(* CODESYS project PresentazioneGIT
   Author: Francesco
   Title: M262 Slave Modbus e ServerOPC_UA
   Version: 0.0.0.0

Project tree, tasks and I/O mapping:
  MyController : TM262L10MESE8T, Schneider Electric, order no. TM262L10MESE8T, version 5.2.8.12
      settings: Enable OPC-UA Server = True; NTP_SERVERENA = False; InterfaceUsedByDhcpSize = 0
    application Application
      libraries: HttpHandling, 1.3.6.0 (Schneider Electric); SysTimeRtc, * (System); TcpUdpCommunication, 2.3.0.0 (Schneider Electric); SysMem, * (System); VisuDialogs, * (System); IecRtsServices, 1.0.5.0 (Schneider Electric); TimeSync, 1.1.7.0 (Schneider Electric); CertificateHandling, 1.2.1.0 (Schneider Electric); CAA File, * (CAA Technical Workgroup)
      task MAST (cyclic, interval 20 ms, priority 15, watchdog 60 ms x 2) calls POU_API_Manuale
      program Certificate_Handling [ST]
      Prog_MatteoLoda/
        data type DUT_result_GET
        global variables GVL_opcua
        global variables PersistentVars
        program POU_API_Manuale [ST]: ACT_Gestione_String_Lettura, New_action
        Symbols
    Diagnostic
    Machine Assistant
    Message Logger
    COM_Bus : COM Bus - TMS, Schneider Electric, version 5.2.8.12
        settings: Network Address = [199, 169, 2, 0]
    DI : Digital Inputs, Schneider Electric, version 5.2.8.12
        input  ibDI_IB0 : BYTE  // IB0
        input  ibDI_IB1 : BYTE  // IB1
    DQ : Digital Outputs, Schneider Electric, version 5.2.8.12
        output q0 : BOOL  // QB0.Q0
        output q1 : BOOL  // QB0.Q1
        output q2 : BOOL  // QB0.Q2
        output q3 : BOOL  // QB0.Q3
        unmapped channels: QB0, QB1
    Ethernet_2 : ETH2, Schneider Electric, version 5.2.8.12
        settings: IPAddress = [192, 168, 8, 19]; SubnetMask = [255, 255, 255, 0]; WebServer = TRUE; FTP Server = TRUE; SoMachine Protocol = TRUE; Modbus Server = TRUE; NetManage Protocol = TRUE; SNMP protocol = TRUE; WebVisu protocol = TRUE; Secured Web Server = TRUE; Remote Connection = TRUE
    Ethernet_Sercos : ETH1, Schneider Electric, version 5.2.8.12
        settings: IPAddress = [192, 168, 1, 91]; SubnetMask = [255, 255, 255, 0]; GatewayAddress = [192, 168, 1, 1]; WebServer = TRUE; FTP Server = TRUE; SoMachine Protocol = TRUE; Modbus Server = TRUE; NetManage Protocol = TRUE; SNMP protocol = TRUE; WebVisu protocol = TRUE; Secured Web Server = TRUE; Remote Connection = TRUE
    IO_Bus : IO bus - TM3, Schneider Electric, version 5.2.8.12
    Serial_Line : Serial line, Schneider Electric, version 5.2.8.12
  5ce3da45-db07-42e7-a21c-a00fff4ed8f6|C:\Users\sesa18348\Downloads\connectivity_1024_768.jpg
  text list GlobalTextList
  function GetCompany [ST]
  function GetTextProperty2 [ST]
  function GetTextProperty [ST]
  function GetTitle [ST]
  function GetVersion [ST]
  function GetVersionProperty [ST]
*)

// MyController/Application/Prog_MatteoLoda/DUT_result_GET
TYPE DUT_result_GET :
STRUCT
	valore:  STRING;
	timestamp:  STRING;
END_STRUCT
END_TYPE

// MyController/Application/Prog_MatteoLoda/GVL_opcua
VAR_GLOBAL
	

scada_data_ora_start : STRING  ;  // data ora start , arriva da scada expert con questo formato : '2023-06-20T04:44:30Z'
scada_data_ora_end : STRING  ; // data ora start , arriva da scada expert con questo formato : '2023-06-20T04:45:00Z' 

Result_Get_value: ARRAY[0..19] OF STRING;
Result_Get_timestamp: ARRAY[0..19] OF STRING;
puntatore_GET: INT;


reset_n_richieste : BOOL ;


ind_IP_Dominio : STRING ; // ip ricevuto da funzione dns
x_dns_OK: BOOL; // dns ok significa anche internet ok
x_dns_ERR: BOOL; // dns err significa anche errore internet
//x_Ping_OK: BOOL;
//x_Ping_ERR: BOOL;
result_HTTP: STRING(INT#15); 
http_client_state			: SE_HTTP.ET_State; // Idle=0, Connecting=10, Connected=20, SendingRequest=30 , Disconnecting=40 ,ResponseAvailable=50 ,Error=-10	
n_dns_ERR: UDINT;

gx_StartCertHandling : bool;


END_VAR

// MyController/Application/Prog_MatteoLoda/PersistentVars

VAR_GLOBAL PERSISTENT RETAIN
	






diag_n_richieste_OK : UDINT ;
diag_n_richieste_ERR : UDINT ;

time_polling : INT ; // tempo base ms












END_VAR

// MyController/Application/Prog_MatteoLoda/POU_API_Manuale
PROGRAM POU_API_Manuale
VAR CONSTANT
String_Unit_ID : ARRAY[0..19] OF STRING := ['formula_ids=2925', 'unit_ids=36389', 'unit_ids=36384', 'unit_ids=36387', 'formula_ids=2931', 'unit_ids=36342', 'unit_ids=36337', 'unit_ids=36340', 'formula_ids=2929', 'unit_ids=36351', 'unit_ids=36346', 'unit_ids=36349', 'formula_ids=2930', 'unit_ids=36371', 'unit_ids=36366', 'unit_ids=36369', 'formula_ids=2928', 'unit_ids=36380', 'unit_ids=36375', 'unit_ids=36378'] ;
END_VAR

VAR
String_Resource: STRING(200);

// Lib usate in questa Demo : SE_HTTP ( x funzioni di connessione e scritture https )
// Lib usate in questa Demo : TCPUDP ( x funzione dns )
// Lib usate in questa Demo : SysTimeRtc ( x funzione timestamp )		
FB_DNSCLIENT				: TCPUDP.FB_DnsClient;			// dichiarazione dell'FB DNS per recupero indirizzo ip del server
FB_HTTP_CLIENT				: SE_HTTP.FB_HttpClient;		// dichiarazione dell'FB CLIENT per connessione , scrittura dati e disconnessione
PARAM_ConnectToServer		: SE_HTTP.TlsSettings;			// ingresso dell'FB : FB_HTTP_CLIENT.ConnectToServer	

Get_Result: SE_HTTP.ET_Result;

Get_result_Msg : STRING ;
Get_Additional_Header: STRING;
Get_Response_Buffer : STRING(5000); // ricezione dati  , per export opcua max(254)
get_error: BOOL;
Get_Strart_request: BOOL;
Get_String_Resource: STRING(SE_HTTP.GPL.Gc_uiMaxLengthOfResource);
FB_PING: TCPUDP.FB_Ping;
ResultPing: STRING(80);
xResultPing: BOOL;
xExecPing : BOOL ;
xResultConnect: SE_HTTP.ET_Result;
temp_string: STRING(1000);
key: STRING(INT#5);
key_stamp: STRING(INT#9);
i: INT;
b: INT;
c: INT;
key2: STRING(INT#1);
a: INT;

x: INT;

	sts: INT;
	sts_prec: INT;
	
	FB_Rit_Start_Polling: TON;
	Dns_leggi_ip: BOOL;
cmd_Reset_Disconnect: BOOL;
cmd_CONNESSIONE: BOOL;
	n_bcd: BYTE;
	FB_NTP: TIMS.FB_SntpClient;
	F_Blink_01: BLINK;
	ntp_manual: BOOL;
	


x_Ping_OK  : BOOL;
x_Ping_ERR : BOOL;

	xNtp_first_time: BOOL;
	xNtp_first_time_done: BOOL;

ritardo_primo_ntp : TON;
impulso_primo_ntp : TP;

ritarda_CertHandling : TON;
END_VAR


// esempio string richiesta GET
// '/api/v2/export/?start=2023-06-20T04:44:30Z&end=2023-06-20T04:45:00Z&unit_ids=36389'
String_Resource := CONCAT('/api/v2/export/?start=',scada_data_ora_start) ; // prepara string get
String_Resource := CONCAT(String_Resource,'&end=') ;// prepara string get
String_Resource := CONCAT(String_Resource,scada_data_ora_end) ;// prepara string get
String_Resource := CONCAT(String_Resource,'&') ;// prepara string get
String_Resource := CONCAT(String_Resource,String_Unit_ID[puntatore_GET]) ;// prepara string get


// parametri per FB connessione
PARAM_ConnectToServer.etProtocol 		:= TCPUDP.ET_TlsProtocol.TLSv13 ;  				// impostazione Parametri per FB seguente 
PARAM_ConnectToServer.etCertVerifyMode 	:= TCPUDP.ET_CertVerifyMode.TrustedOnly  ;	 	// impostazione Parametri per FB seguente

// parametri per FB GET
//Get_String_Resource := '/api/v2/export/?start=2023-06-20T04:44:30Z&end=2023-06-20T04:45:00Z&unit_ids=36389'   ; // 
Get_String_Resource := String_Resource  ; // 
Get_Additional_Header :=  'Authorization: Basic emVudHJpeDpyaXZlcmxha2U='   ; // 'Authorization: Basic b3BlcmF0b3I6ZGU0NzU5MzE='  codificato in base64
	



//---------------------------------------------------------------------------------------------------------------------

// time_polling
IF time_polling<5 THEN // timepolling è usato come ritardo tra richieste , tempo min 5 ms
	time_polling := 5 ; // tempo min 5 ms
END_IF
FB_Rit_Start_Polling(
	IN:=NOT Dns_leggi_ip , 
	PT:= INT_TO_TIME(time_polling), 
	Q=> , 
	ET=> );
IF 	FB_Rit_Start_Polling.Q THEN
	Dns_leggi_ip:=TRUE;
END_IF

//---------------------------------------------------------------------------------------------------------------------

FB_DNSCLIENT(
	i_xEnable			:=  Dns_leggi_ip, 
	i_xExecute			:=  FB_DNSCLIENT.q_xActive AND FB_DNSCLIENT.q_xReady, 
	i_sDnsServerIP		:= '8.8.8.8', // dns di google
	i_uiDnsServerPort	:= , 
	i_sDomainName		:=  'ehp-data.com',  // dominio
	q_xActive			=> , 
	q_xReady			=> , 
	q_xBusy				=> , 
	q_xDone				=> x_dns_OK, 
	q_xError			=> x_dns_ERR, 
	q_etResult			=> , 
	q_sResultMsg		=> , 
	q_uiNumberOfIpAddresses	=> , 
	q_astDnsAddressInfo		=> ); // in questo (.q_astDnsAddressInfo[0].sIpAddress) l'indirizzo IP del server
		

IF FB_DNSCLIENT.q_xDone THEN
	ind_IP_Dominio := FB_DNSCLIENT.q_astDnsAddressInfo[0].sIpAddress	;
	xExecPing := TRUE ;

END_IF
IF FB_DNSCLIENT.q_xError THEN
	Dns_leggi_ip := FALSE ;
	n_dns_ERR := n_dns_ERR +1 ;
END_IF


	
// se abilito il ping il polling ritarda causa esecuzione del ping
FB_PING(
	i_xExecute:= xExecPing, 
	i_sDeviceIP:= ind_IP_Dominio , // '135.181.0.23'
	i_timTimeout:= T#5S, 
	q_xBusy=> , 
	q_xDone=> x_Ping_OK, 
	q_xError=> x_Ping_ERR, 
	q_etResult=> , 
	q_sResultMsg=> ResultPing);

IF x_Ping_OK THEN
	gx_StartCertHandling:=TRUE;
END_IF
ritarda_CertHandling(in:=gx_StartCertHandling, pt:=T#500MS);
IF ritarda_CertHandling.Q THEN
	Certificate_Handling();
END_IF


//---------------------------------------------------------------------------------------------------------------------
IF FB_DNSCLIENT.q_xDone THEN // x_Ping_OK
	cmd_CONNESSIONE := TRUE ;
END_IF
http_client_state :=  FB_HTTP_CLIENT.State ;

IF cmd_CONNESSIONE AND FB_HTTP_CLIENT.State = SE_HTTP.ET_State.Idle THEN 			
	FB_HTTP_CLIENT.ConnectToServer(
		i_sServerIP			:= ind_IP_Dominio , // Indirizzo_IP_server   '135.181.0.23' 
		i_uiServerPort		:= 443 , //443
		i_xUseTls			:= TRUE , // true con port 443 , false per port 80
		i_stTlsSettings		:= PARAM_ConnectToServer, 
		q_xError	=> , 
		q_etResult	=>  xResultConnect, 
		q_sResultMsg=> );
END_IF

IF FB_HTTP_CLIENT.State=SE_HTTP.ET_State.Connected THEN
	FB_HTTP_CLIENT.Get( 
		i_sResource := Get_String_Resource ,
		i_sHost:= 'ehp-data.com' ,// ehp-data.com
		i_anyAdditionalHeader:= Get_Additional_Header, // string Header    'Authorization: Basic b3BlcmF0b3I6ZGU0NzU5MzE='
		i_anyResponseBuffer:= Get_Response_Buffer, // string_xy.000 // ricezione dati
		q_xError=> get_error, 
		q_etResult=> Get_Result , 
		q_sResultMsg=> Get_result_Msg );	
END_IF


ACT_Gestione_String_Lettura();




//---------------------------------------------------------------------------------------------------------------------
IF cmd_Reset_Disconnect OR FB_HTTP_CLIENT.State = SE_HTTP.ET_State.Error THEN
	FB_HTTP_CLIENT.DisconnectFromServer(
		q_xError=> , 
		q_etResult=> , 
		q_sResultMsg=> );
	FB_HTTP_CLIENT.Reset();
	cmd_Reset_Disconnect := FALSE ;
	get_error := FALSE ;
	Dns_leggi_ip := FALSE ;
	xExecPing := FALSE ;
	cmd_CONNESSIONE := FALSE ;
	Get_Strart_request := FALSE ;
	Get_Response_Buffer:='';
	Get_Additional_Header:='';
	Get_result_Msg:='';
	puntatore_GET := puntatore_GET +1 ;
	IF puntatore_GET>19 THEN
		puntatore_GET:=0;
	END_IF
END_IF



n_bcd := int_to_bcd(puntatore_GET); // sposto valore puntatore in uscite plc formato bcd
q0:= n_bcd.0 ; // uscita plc
q1:= n_bcd.1 ;// uscita plc
q2:= n_bcd.2 ;// uscita plc
q3:= n_bcd.3 ;// uscita plc



IF reset_n_richieste THEN
	diag_n_richieste_OK := 0 ;
	diag_n_richieste_ERR := 0;
	n_dns_ERR:=0;
	reset_n_richieste := FALSE ;
END_IF

F_Blink_01(ENABLE:=TRUE , TIMELOW:=T#10M , TIMEHIGH:=T#5S , OUT=> );

ritardo_primo_ntp(IN:= NOT xNtp_first_time_done, PT:= T#30S, Q=> , ET=> );
impulso_primo_ntp(IN:= ritardo_primo_ntp.Q, PT:= T#1S, Q=> xNtp_first_time, ET=> );
IF xNtp_first_time THEN
	xNtp_first_time_done:=TRUE;
END_IF

FB_NTP.i_stTimeRequest.i_sServerIp := '95.217.220.251' ;
FB_NTP.i_stTimeRequest.i_timServerTimeOut := T#3000MS;
FB_NTP(
	i_xEnable:= F_Blink_01.OUT OR ntp_manual OR xNtp_first_time, //
	i_xExecute:= FB_NTP.q_xActive AND FB_NTP.q_xReady, 
	i_xSyncRtc:= TRUE, 
	i_diTimeZone:= , 
	i_uiMaxRtcOffset:= , 
	i_stTimeRequest:= , 
	q_xActive=> , 
	q_xReady=> , 
	q_xBusy=> , 
	q_xDone=> , 
	q_stTimeResponse=> , 
	q_xError=> , 
	q_etResult=> , 
	q_sResultMsg=> );

ACTION ACT_Gestione_String_Lettura:





//temp_string:='HTTP/1.1 200 OK$R$NDate: Fri, 26 Jan 2024 10:04:06 GMT$R$NContent-TYPE: application/json$R$NServer: gunicorn/19.6.0$R$NVary: Accept, Accept-Language, Cookie$R$NContent-Language: en$R$NAllow: OPTIONS, GET$R$NTransfer-Encoding: chunked$R$NConnection: keep-alive$R$N$R$Ncd$R$N{"count":1,"previous":null,"results":[{"timestamp":"2023-06-20T04:45:00Z","value":6.196179294586182,"raw":true,"formula":null,"id":1375400206,"unit":"http://ehp-data.com/api/v2/units/36389/"}],"next":null}$R$N0$R$N$R$N';
temp_string := Get_Response_Buffer ;

FOR x:=0 TO 15 DO 
	result_HTTP[x]:= temp_string[x];
END_FOR


result_HTTP :=result_HTTP ;

IF result_HTTP ='HTTP/1.1 200 OK' THEN
	i:=0;
	key:='';
	WHILE key<>'value' DO
		key[0+0]:= temp_string[i+0];
		key[0+1]:= temp_string[i+1];
		key[0+2]:= temp_string[i+2];
		key[0+3]:= temp_string[i+3];
		key[0+4]:= temp_string[i+4];
		i:=i+1;
		b:=i+6;
		IF i >= 400 THEN
			EXIT;
		END_IF
	END_WHILE
	
	
	a:=0;
	key2:='';
	WHILE key2<>',' DO // la virgola è 44 in decimale
		key2[0]:= temp_string[b+a];
		a:=a+1;
		c:=a;
		IF a >= 400 THEN
			EXIT;
		END_IF
	END_WHILE
	
	
	Result_Get_value[puntatore_GET] := '';
	IF key2=','  AND key='value' THEN
		FOR x:=b TO b+c-2 DO 
			Result_Get_value[puntatore_GET][x-b]:= temp_string[x];
		END_FOR	
	END_IF
	
	
	//FG------------------------------------------------
	i:=0;
	key_Stamp:='';
	WHILE key_Stamp<>'timestamp' DO
		key_Stamp[0+0]:= temp_string[i+0];
		key_Stamp[0+1]:= temp_string[i+1];
		key_Stamp[0+2]:= temp_string[i+2];
		key_Stamp[0+3]:= temp_string[i+3];
		key_Stamp[0+4]:= temp_string[i+4];
		key_Stamp[0+5]:= temp_string[i+5];
		key_Stamp[0+6]:= temp_string[i+6];
		key_Stamp[0+7]:= temp_string[i+7];
		key_Stamp[0+8]:= temp_string[i+8];
		i:=i+1;
		b:=i+11;
		IF i >= 400 THEN
			EXIT;
		END_IF
	END_WHILE
	a:=0;
	key2:='';
	WHILE key2<>',' DO // la virgola è 44 in decimale
		key2[0]:= temp_string[b+a];
		a:=a+1;
		c:=a;
		IF a >= 400 THEN
			EXIT;
		END_IF
	END_WHILE
	
	Result_Get_timestamp[puntatore_GET] := '';
	IF key2=','  AND key_Stamp='timestamp' THEN
		FOR x:=b TO b+c-3 DO 
			Result_Get_timestamp[puntatore_GET][x-b]:= temp_string[x];
		END_FOR	
	END_IF
	
	//FG-----------------------------------------------------------------
	
	//string_valore ;
	cmd_Reset_Disconnect:=TRUE;
	diag_n_richieste_OK := diag_n_richieste_OK +1 ;
END_IF



IF result_HTTP <>'HTTP/1.1 200 OK' AND result_HTTP <>'' THEN
	cmd_Reset_Disconnect:=TRUE;
	diag_n_richieste_ERR := diag_n_richieste_ERR +1 ;
END_IF
END_ACTION

ACTION New_action:
//ho inserito un nuovo blocco di codice
END_ACTION

END_PROGRAM

// MyController/Application/Certificate_Handling
PROGRAM Certificate_Handling
VAR
// 	open : file.diropen;
// 	close: file.DirClose;
// 	copy : file.DirCopy;
// 	remove_quarantena: file.DirRemove;
// 	remove_trusted: file.DirRemove;
	
FB_CH : se_cert.FB_CertificateHandling;
F_Blink_Certificate: BLINK;
xDoneSCT : BOOL;
xDoneSCQ : BOOL;
xDoneC : BOOL;
xDoneDT : BOOL;
xDoneDQ : BOOL;

xErrorSCT : BOOL;
xErrorSCQ : BOOL;
xErrorC : BOOL;
xErrorDT : BOOL;
xErrorDQ : BOOL;

xBusy :BOOL;

udicase: INT;
risultato_comunicazione : se_cert.et_result;
stato_comunicazione :  se_cert.et_state;
END_VAR

// //------------------------------------------------------------------------
// 
// F_Blink_Certificate(ENABLE:=TRUE , TIMELOW:=T#10S , TIMEHIGH:=T#5S , OUT=> );//F_Blink_Certificate(ENABLE:=TRUE , TIMELOW:=T#1D , TIMEHIGH:=T#5S , OUT=> );
// IF F_Blink_Certificate.out THEN
// 	//seleziono il certificato e lo copio nei trusted
// 	IF FB_CH.SelectFirstCertificate(i_etTrustLevel:= 3, i_timTimeout:= T#10S, q_xBusy=> , q_xDone=> xCertificateSelection, q_xError=> ) THEN//c'è qualcosa in quarantena?
// 	
// 		IF FB_CH.SelectFirstCertificate(i_etTrustLevel:= 1, i_timTimeout:= T#10S, q_xBusy=> , q_xDone=> xCertificateSelection, q_xError=> )	THEN//pulisco i trusted
// 			 FB_CH.Delete(i_timTimeout:= T#5S, q_xBusy=> , q_xDone=> , q_xError=> );
// 		END_IF
// 		IF FB_CH.SelectFirstCertificate(i_etTrustLevel:= 3, i_timTimeout:= T#10S, q_xBusy=> , q_xDone=> xCertificateSelection, q_xError=> ) THEN
// 			IF FB_CH.Copy(i_etDestinationTrustLevel:= 1, i_timTimeout:= T#10S, q_xBusy=> , q_xDone=> xCertificateCopy, q_xError=> ) THEN //copio in trusted
// 				IF FB_CH.SelectFirstCertificate(i_etTrustLevel:= 3, i_timTimeout:= T#10S, q_xBusy=> , q_xDone=> xCertificateSelection, q_xError=> ) THEN
// 					FB_CH.Delete(i_timTimeout:= T#5S, q_xBusy=> , q_xDone=> , q_xError=> );														//elimino dalla quarantena
// 				END_IF
// 			END_IF
// 		END_IF
// 	END_IF
// END_IF


IF udicase=0 THEN
	FB_CH.SelectFirstCertificate(i_etTrustLevel:= 3, i_timTimeout:= T#10S, q_xBusy=> xBusy, q_xDone=> xDoneSCQ, q_xError=> xErrorSCQ);
	IF xDoneSCQ THEN
		udicase:=5;
	END_IF
	IF xErrorSCQ THEN
		udicase:=1000;
	END_IF
END_IF

IF udicase=5 THEN
	IF fb_ch.IsCertificateSelected THEN
		udicase:=10;
	END_IF
END_IF

IF udicase =10 THEN
	FB_CH.SelectFirstCertificate(i_etTrustLevel:= 1, i_timTimeout:= T#10S, q_xBusy=> , q_xDone=> xDoneSCT, q_xError=> xErrorSCT);
	IF xDoneSCT OR  xErrorSCT THEN
		IF fb_ch.IsCertificateSelected THEN
			udicase:=12;
		ELSE
			IF FB_CH.ReleaseCertificate() THEN
				udicase:=20;
			END_IF
		END_IF
	END_IF
END_IF

IF udicase =12 THEN
	FB_CH.Delete(i_timTimeout:= T#10S, q_xBusy=> , q_xDone=> xDoneDT, q_xError=> xErrorDT);
	IF xDoneDT OR  xErrorDT THEN
		udicase:=10;
	END_IF
END_IF



IF udicase =20 THEN
	FB_CH.SelectFirstCertificate(i_etTrustLevel:= 3, i_timTimeout:= T#10S, q_xBusy=> , q_xDone=> xDoneSCQ, q_xError=> xErrorSCQ);
	IF xDoneSCQ OR  xErrorSCQ THEN
		udicase:=25;
	END_IF
END_IF	

IF udicase=25 THEN
	IF fb_ch.IsCertificateSelected THEN
		FB_CH.Copy(i_etDestinationTrustLevel:= 1, i_timTimeout:= T#10S, q_xBusy=> , q_xDone=> xDoneC, q_xError=> xErrorC);
		IF xDoneC OR xErrorC THEN
			 udicase:=27;
		END_IF
	END_IF
END_IF

IF udicase=27 THEN
	IF FB_CH.ReleaseCertificate() THEN
		udicase:=30;
	END_IF
END_IF

			
			
IF udicase =30 THEN
	FB_CH.SelectFirstCertificate(i_etTrustLevel:= 3, i_timTimeout:= T#10S, q_xBusy=> , q_xDone=> xDoneSCQ, q_xError=> xErrorSCQ);
	IF xDoneSCQ OR xErrorSCQ THEN
		udicase :=35;
	END_IF
END_IF

IF udicase =35 THEN
	FB_CH.Delete(i_timTimeout:= T#10S, q_xBusy=> , q_xDone=> xDoneDQ, q_xError=> xErrorDQ);
	IF xDoneDQ OR xErrorDQ THEN
		IF FB_CH.ReleaseCertificate() THEN
			udicase:=0;
		END_IF
	END_IF	
END_IF


IF udicase =1000 THEN
	 udicase :=0;
END_IF

END_PROGRAM

// GetCompany
// This function has been automatically generated from the project information.
{attribute 'signature_flag' := '1073741824'}
{attribute 'register_in_runtime'}
FUNCTION GetCompany : WSTRING
VAR_INPUT
	
END_VAR

GetCompany := "";

END_FUNCTION

// GetTextProperty2
// This function has been automatically generated from the project information.
{attribute 'signature_flag' := '1073741824'}
{attribute 'register_in_runtime'}
FUNCTION GetTextProperty2 : POINTER TO WSTRING
VAR_INPUT
	stKey: WSTRING;
END_VAR

IF stKey = "Author" THEN
	GetTextProperty2 := ADR("Francesco");
ELSIF stKey = "Company" THEN
	GetTextProperty2 := ADR("");
ELSIF stKey = "Description" THEN
	GetTextProperty2 := ADR("");
ELSIF stKey = "Project" THEN
	GetTextProperty2 := ADR("Test");
ELSIF stKey = "Title" THEN
	GetTextProperty2 := ADR("M262 Slave Modbus e ServerOPC_UA");
ELSE
	GetTextProperty2 := ADR("");
END_IF

END_FUNCTION

// GetTextProperty
// This function has been automatically generated from the project information.
{attribute 'signature_flag' := '1073741824'}
{attribute 'register_in_runtime'}
FUNCTION GetTextProperty : WSTRING
VAR_INPUT
	stKey: WSTRING;
END_VAR

IF stKey = "Author" THEN
	GetTextProperty := "Francesco";
ELSIF stKey = "Company" THEN
	GetTextProperty := "";
ELSIF stKey = "Description" THEN
	GetTextProperty := "";
ELSIF stKey = "Project" THEN
	GetTextProperty := "M262 API_GET_HANNUKAINEN_https_ntp_dns_get_V13";
ELSIF stKey = "Title" THEN
	GetTextProperty := "M262 Slave Modbus e ServerOPC_UA";
ELSE
	GetTextProperty := "";
END_IF

END_FUNCTION

// GetTitle
// This function has been automatically generated from the project information.
{attribute 'signature_flag' := '1073741824'}
{attribute 'register_in_runtime'}
FUNCTION GetTitle : WSTRING
VAR_INPUT
	
END_VAR

GetTitle := "M262 Slave Modbus e ServerOPC_UA";

END_FUNCTION

// GetVersion
// This function has been automatically generated from the project information.
{attribute 'signature_flag' := '1073741824'}
{attribute 'register_in_runtime'}
FUNCTION GetVersion : VERSION
VAR_INPUT
	
END_VAR

GetVersion.uiMajor := 0;
GetVersion.uiMinor := 0;
GetVersion.uiServicePack := 0;
GetVersion.uiPatch := 0;

END_FUNCTION

// GetVersionProperty
// This function has been automatically generated from the project information.
{attribute 'signature_flag' := '1073741824'}
{attribute 'register_in_runtime'}
FUNCTION GetVersionProperty : VERSION
VAR_INPUT
	stKey: WSTRING;
END_VAR

IF stKey = "Version" THEN
	GetVersionProperty.uiMajor := 0;
	GetVersionProperty.uiMinor := 0;
	GetVersionProperty.uiServicePack := 0;
	GetVersionProperty.uiPatch := 0;
ELSE
	GetVersionProperty.uiMajor := 0;
	GetVersionProperty.uiMinor := 0;
	GetVersionProperty.uiServicePack := 0;
	GetVersionProperty.uiPatch := 0;
END_IF

END_FUNCTION
